// TIA Portal V19 export
DATA_BLOCK "Production_HMI"   // DB9
// stored: MemoryReserve 100
   VAR
      MAN_O : Struct
         PPrf_No : DInt;
         Req : DInt;
         Len : Real;
         Use_Ribbing_Roll : Bool;
         Use_Trace_Mark_Tool : Bool;
         Use_Thick_Mark_Tool : Bool;
      END_STRUCT;
      Sel_Index : Int;   // Riga degli ordini da fare selezionata
      Button_Pop_ACT_To_ENDING : Struct   // Pulsante HMI per spostare ordine al taglio completato su ordini in via di completamento
         Show : Bool;
         AllowControl : Bool;
         Pressed : Bool;
         Done { ExternalAccessible := 'False'; ExternalVisible := 'False'; ExternalWritable := 'False'} : Bool;
         Error { ExternalAccessible := 'False'; ExternalVisible := 'False'; ExternalWritable := 'False'} : Bool;
         Color : Int;
      END_STRUCT;
      Button_Pop_ACT_To_TODO : Struct   // Pulsante HMI per interrompere ordine al taglio non completato su lista ordini da fare
         Show : Bool;
         AllowControl : Bool;
         Pressed : Bool;
         Done { ExternalAccessible := 'False'; ExternalVisible := 'False'; ExternalWritable := 'False'} : Bool;
         Error { ExternalAccessible := 'False'; ExternalVisible := 'False'; ExternalWritable := 'False'} : Bool;
         Color : Int;
      END_STRUCT;
      Button_Pop_TODO_To_ACT : Struct   // Pulsante HMI per spostare in lavoro l'ordine selezionato dalla lista di quelli da fare
         Show : Bool;   // Abiliita visualizzazione button che avvia il comando
         AllowControl : Bool;   // Abilita pulsanti nascosti di selezione riga
         Pressed : Bool;   // Set con pulsante premuto, Rst da PLC
         Done : Bool;
         Error : Bool;
         Color : Int;
      END_STRUCT;
      Button_Push_ManualOrder_To_TODO : Struct   // Gestione Pulsante HMI per caricamento ordine manuale su lista ordini da fare
         Show : Bool;
         AllowControl : Bool;
         Pressed : Bool;
         Done : Bool;
         Error : Bool;
         Color : Int;
      END_STRUCT;
      Buttons_ChangeOrder_TODO : Struct   // Gestione Pulsanti HMI per cambiare ordine di esecuzione della lista ordini da fare (Solo se MES è OFF)
         Show : Bool;   // Abiliita visualizzazione button che avvia il comando
         AllowControl : Bool;   // Abilita pulsanti nascosti di selezione riga
         Pressed_UP : Bool;   // (Set con pulsante premuto, Rst da PLC) Sposta in alto (indice più piccolo)
         Pressed_DW : Bool;   // (Set con pulsante premuto, Rst da PLC) Sposta in basso (indice più grande)
      END_STRUCT;
      Button_Pop_TODO_To_ENDING : Struct   // Gestione Pulsante HMI per sposatre ordine di lavoro da in esecuzione a in via di completamento (solo se MES è OFF)
         Show : Bool;   // Abiliita visualizzazione button che avvia il comando
         AllowControl : Bool;   // Abilita pulsanti nascosti di selezione riga
         Pressed : Bool;   // Set con pulsante premuto, Rst da PLC
         Done : Bool;
         Error : Bool;
         Color : Int;
      END_STRUCT;
      Button_ShowDetatails : Struct   // Pulsante HMI per spostare ordine al taglio completato su ordini in via di completamento
         Show : Bool;
         Pressed : Bool;
         Data { S7_SetPoint := 'True'} : "Prod_Item";
      END_STRUCT;
      SETUP : Struct   // Gestione SETUP operazini manuali
         Button_LinePreparation_Start : Struct   // Gestione Pulsante HMI per sposatre ordine di lavoro da in esecuzione a in via di completamento (solo se MES è OFF)
            Show : Bool;   // Abiliita visualizzazione button che avvia il comando
            AllowControl : Bool;   // Abilita pulsanti nascosti di selezione riga
            Pressed : Bool;   // Set con pulsante premuto, Rst da PLC
            Done : Bool;
            Error : Bool;
            Color : Int;
         END_STRUCT;
         Button_LinePreparation_Stop : Struct   // Gestione Pulsante HMI per sposatre ordine di lavoro da in esecuzione a in via di completamento (solo se MES è OFF)
            Show : Bool;   // Abiliita visualizzazione button che avvia il comando
            AllowControl : Bool;   // Abilita pulsanti nascosti di selezione riga
            Pressed : Bool;   // Set con pulsante premuto, Rst da PLC
            Done : Bool;
            Error : Bool;
            Color : Int;
         END_STRUCT;
         Button_OP_Man_X_Pressed : Array[1.."SETUP_MAN_OPERATIONS_QTY"] of Bool;   // Bit usato come "on con tasto premuto" - ACK op.man.con su array REAL
         Button_OP_Man_Y_Pressed : Array[1.."SETUP_MAN_OP_WITH_CODE_QTY"] of Bool;   // Bit usato come "on con tasto premuto" - ACK op.man.con su array INT
         Button_OP_Man_Z_Pressed : Array[1.."PROD_SETUP_WAIT_MAN_PREPARATION"] of Bool;   // Bit usato come "on con tasto premuto" - ACK op.man.con su array INT
         Button_OP_Man_Set_All_OK : Struct   // Pulsante HMI per impostare OK su tutte le operazioni manuali
            Show : Bool;
            AllowControl : Bool;
            Pressed : Bool;
            Done { ExternalAccessible := 'False'; ExternalVisible := 'False'; ExternalWritable := 'False'} : Bool;
            Error { ExternalAccessible := 'False'; ExternalVisible := 'False'; ExternalWritable := 'False'} : Bool;
            Color : Int;
         END_STRUCT;
         "SetUp_OP-Man_OK_Cumultativo" : Bool;
         SetUp_OP_Man_X_OK : Array[1.."SETUP_MAN_OPERATIONS_QTY"] of Bool;
         SetUp_OP_Man_Y_OK : Array[1.."SETUP_MAN_OP_WITH_CODE_QTY"] of Bool;
         SetUp_Aut_Profilatrice_OK_Cumultativo : Bool;
         SetUp_Aut_Bordatrice_OK_Cumultativo : Bool;
         SetUp_Aut_OK_Profilatrice : Array[1..14] of Bool;   // Stati del singolo asse di preparazione della PROFILATRICE in posizione richiesta per setup
         SetUp_Aut_OK_Bordatrice : Array[1..9] of Bool;   // Stati del singolo asse di preparazione della BORDATRICE in posizione richiesta per setup
      END_STRUCT;
      Material_To_GO_Cumulative : LReal;
      OrdineKanban_Presence { S7_SetPoint := 'True'} : Bool;
      StampoTracciabilita_Attuale : Struct
         IDRotolo : String;
         NumeroColata : String;
      END_STRUCT;
      StampoTracciabilita_Prossimo : Struct
         IDRotolo : String;
         NumeroColata : String;
      END_STRUCT;
   END_VAR
BEGIN
END_DATA_BLOCK
